// TIA Portal project "Cau3" (V16)

(* hardware
DEVICE "S7-1200 station_1"  S7-1200 Station
   slot 0: "Rack_0"  S7-1200 Rack  Rack  V1.0
   slot 1: "PLC_1"  CPU 1212C DC/DC/DC  6ES7 212-1AE40-0XB0  V4.3
   slot 2: "DI 16/DQ 16x24VDC_1"  6ES7 223-1BL32-0XB0  V2.0
   slot 3: "DQ 16xRelay_1"  SM 1222 DQ16 x relay  6ES7 222-1HH32-0XB0  V2.0
*)

// ===== PLC "PLC_1"  CPU 1212C DC/DC/DC =====

VAR_GLOBAL   // PLC tag table "Default tag table"
   "Stop" AT %I8.2 : Bool;
   "Start" AT %I8.3 : Bool;
   "Biến giữ KM5 + KM7" AT %M0.0 : Bool;
   "KM6" AT %Q0.5 : Bool;
   "KM7" AT %Q1.1 : Bool;
   "KM5" AT %Q0.4 : Bool;
END_VAR

// folder: System blocks/Program resources

DATA_BLOCK "T1"   // DB1
{ S7_Optimized_Access := 'TRUE' }
AUTHOR : Simatic
FAMILY : IEC
NAME : IEC_TMR
VERSION : 1.0
// stored: InstanceOfName IEC_TIMER
"IEC_TIMER"
BEGIN
END_DATA_BLOCK

// folder: (top level)

ORGANIZATION_BLOCK "Main"   // OB1, LAD, ProgramCycle
TITLE = "Main Program Sweep (Cycle)"
{ S7_Optimized_Access := 'TRUE' }
VERSION : 0.1
   VAR_INPUT
      Initial_Call : Bool;   // Initial call of this OB
      Remanence : Bool;   // =True, if remanent data are available
   END_VAR
BEGIN

REGION Network 1
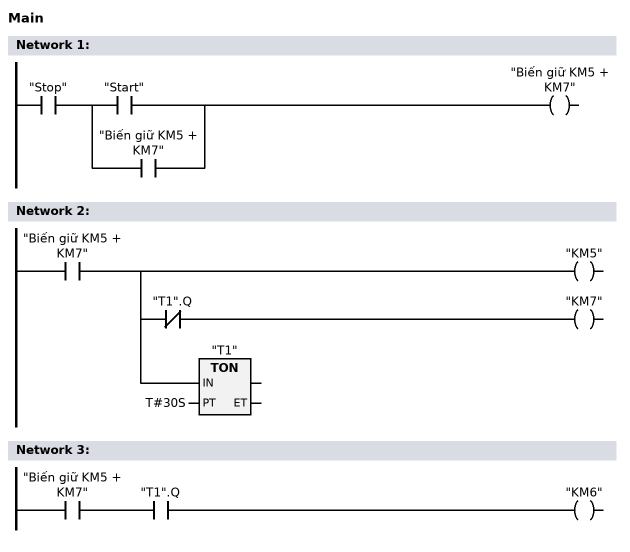
   RUNG wire#powerrail
      Contact( "Stop" )
      wire#w1
      Contact( "Start" )
      wire#w2
      Coil( "Biến giữ KM5 + KM7" )
   END_RUNG
   RUNG wire#w1
      Contact( "Biến giữ KM5 + KM7" )
   END_RUNG wire#w2
   // the same network as SCL:
   "Biến giữ KM5 + KM7" := "Stop" AND ("Start" OR "Biến giữ KM5 + KM7");
END_REGION

REGION Network 2
   "KM5" := "Biến giữ KM5 + KM7";
   "KM7" := "Biến giữ KM5 + KM7" AND NOT "T1".Q;
   "T1".TON(IN := "Biến giữ KM5 + KM7", PT := T#30S);
END_REGION

REGION Network 3
   RUNG wire#powerrail
      Contact( "Biến giữ KM5 + KM7" )
      Contact( "T1".Q )
      Coil( "KM6" )
   END_RUNG
   // the same network as SCL:
   "KM6" := "Biến giữ KM5 + KM7" AND "T1".Q;
END_REGION
END_ORGANIZATION_BLOCK